(* IEC 61131-3 sources: std_i2980_v2.06_cp053/Source/IMM/ieccontrol/system, 15 files *)

(* ---- ABCfgLoader.pu ---- *)
(*
@h    ! WARNING !
@h    The Kemro K2 system (including software) only meets category B according to EN 954-1,
@h    thus it is not intended for usage in safety-relevant control applications in the field
@h    of personal safety (e.g. emergency stop).
@h    To implement potentially necessary safety-relevant control tasks, always use additional
@h    external safety devices that are intended for the particular purpose, and meet the necessary
@h    functional safety.
@h    For further information see EN 954-1 (EN ISO 13849-1) and/or the K2-x00 user manual, chapter
@h    "CE conformity, directives and standards".

This algorithm block reading configuration settings from
the catalogue and copies the values to the according systemvariables.
Reading starts after device registration is completed.
After reading the settings the file appco.cfg is deleted.
*)

IMPORT_OVER_LISTFILE
 KCAT_GetHandle
, FConfigNode
, KCAT_GetValue
, KFILE_Delete
, FCreateIECVersion
, FCreateIECLibVersion
, FCreateIECBaseVersion
, FCreateSystemName
, FCreateHMIKVSVersion
, FCreateHMIStyleVersion
, KSYS_BPAPI_VAR_TXTREAD
, KCAT_Status_OK
, KCAT_Status
, KSYS_BPApiState
, KCAT_HandleData
, KFILE_Status

END_IMPORT

ALGORITHM_BLOCK ABCfgLoader #DUMMY_EDIT_BLOCK

SYSTEM_VAR
 sv_bReadConfigDone : BOOL;
 sv_bDeviceRegisterDone : BOOL;
 sv_bInitStart : BOOL;
 sv_sPathMasterdisk : STRING(255);
 sv_sPathWorkspace : STRING(255);
 sv_sPathAppldisk : STRING(255);
END_VAR

SYSTEM_OBJECT
 TaskMid : TASK;
 PU_Task_7 : TASK;
 TaskSlow : TASK;
END_OBJECT

FUNCTION fCreateOSVersion : BOOL
 #DUMMY_EDIT_BLOCK

VAR
 Status : KCAT_Status;
 SysState : KSYS_BPApiState;
 HandleData : KCAT_HandleData;
 sValue : STRING(255);
 sTmp : STRING(255);
 bLinux : BOOL;
END_VAR
#BEGIN_EDIT_BLOCK
(**************************************** WARNING ********************************************
 *** The KEBA Kemro K2 System including software is not intended for safety control tasks! ***
 ***                       For further information see Comment tab!                        ***
 *********************************************************************************************)

// create extended OS version information in catalog (on Linux systems only)
// necessary for systems like KVS to access OS specific version info without SysRPC/BPAPI

HandleData := KCAT_GetHandle('UOS.System');
IF HandleData.Status = KCAT_Status_OK THEN
   Status := KCAT_GetValue(Handle := HandleData.Handle, Buffer := sValue);
   IF (sValue = 'Linux') THEN
      bLinux := TRUE;
   END_IF;
END_IF;

IF(NOT bLinux) THEN
   // do not create the nodes on VxWorks - this info does not exist
   RETURN;
END_IF;

HandleData := KCAT_GetHandle('System');
IF HandleData.Status <> KCAT_Status_OK THEN
   RETURN;
END_IF;

HandleData := KCAT_AddDir(HandleData.Handle, 'OS');
IF HandleData.Status <> KCAT_Status_OK THEN
   RETURN;
END_IF;

// add device driver version

SysState := KSYS_BPAPI_VAR_TXTREAD('SYS.HW.OS.driversVersion', sValue);
Status := KCAT_AddValue(HandleData.Handle, "driversVersion", KCAT_Type_STRING, sValue);
IF Status <> KCAT_Status_OK THEN
   RETURN;
END_IF;

// add OS specific version (concated)
SysState := KSYS_BPAPI_VAR_TXTREAD('SYS.HW.OS.osType', sTmp);
sValue := CONCAT(sTmp, ' ');

SysState := KSYS_BPAPI_VAR_TXTREAD('SYS.HW.OS.osVersion', sTmp);
sValue := CONCAT(sValue, sTmp, ' ');

SysState := KSYS_BPAPI_VAR_TXTREAD('SYS.HW.OS.kernelVersion', sTmp);
sValue := CONCAT(sValue, sTmp);

Status := KCAT_AddValue(HandleData.Handle, "osVersion", KCAT_Type_STRING, sValue);
IF Status <> KCAT_Status_OK THEN
   RETURN;
END_IF;

fCreateOSVersion := TRUE;

;#END_EDIT_BLOCK END_FUNCTION

PROCESS_ALGORITHM paReadConfig ON TaskMid

VAR
 HandleData : KCAT_HandleData;
 sRootPath : STRING(255);
 // sPath : STRING(255);
 // Status : KCAT_Status;
 // sBasePath : STRING(255);
 fileState : KFILE_Status;
 StatusName_CAT : KCAT_HandleData;
 Status_CAT : KCAT_Status;
END_VAR
#BEGIN_EDIT_BLOCK
(**************************************** WARNING ********************************************
 *** The KEBA Kemro K2 System including software is not intended for safety control tasks! ***
 ***                       For further information see Comment tab!                        ***
 *********************************************************************************************)

//check if data is available
sRootPath := "Application.Application1";
HandleData:=KCAT_GetHandle(sRootPath);
IF HandleData.Status<>KCAT_Status_OK THEN
   //no catalog entries for appliaction available
   sv_bReadConfigDone := TRUE;
   STOP_PROCESS_ALGORITHM();
   RETURN;
END_IF;

(*
//-----------------------------------------------------------
//read actuation params
//-------------------------------------------------------------
sBasePath := CONCAT(sRootPath, ".Actuation");

sPath := CONCAT(sBasePath, ".System_pressure");
Status := FConfigNode(sPath, "system.sv_rMaximumPressure", 1);

sPath := CONCAT(sBasePath, ".System_velocity");
Status := FConfigNode(sPath, "Injection1.sv_rMaxSpeedFwd", 1);

//-------------------------------------------------------------------
//read clamp side parameters
//-------------------------------------------------------------------
sBasePath := CONCAT(sRootPath, ".Closure_unit");

//mold stroke
sPath := CONCAT(sBasePath, ".Stroke_mold");
Status := FConfigNode(sPath, "Mold1.sv_rMoldStroke", 1);

//profile stages mold close
sPath := CONCAT(sBasePath, ".No_profile_points_mold_close");
Status := FConfigNode(sPath, "Mold1.sv_MoldFwdProfVisSrc.Profile.iNoOfPoints", 0);

//profile stages mold open
sPath := CONCAT(sBasePath, ".No_profile_points_mold_open");
Status := FConfigNode(sPath, "Mold1.sv_MoldBwdProfVis.Profile.iNoOfPoints", 0);

//ejector stroke
sPath := CONCAT(sBasePath, ".Stroke_ejector");
Status := FConfigNode(sPath, "Ejector1.sv_rEjectorStroke", 1);

//profile stages ejector bwd
sPath := CONCAT(sBasePath, ".No_profile_points_ejector_bwd");
Status := FConfigNode(sPath, "Ejector1.sv_EjectorBwdVis.Profile.iNoOfPoints", 0);

//profile stages ejector fwd
sPath := CONCAT(sBasePath, ".No_profile_points_ejector_fwd");
Status := FConfigNode(sPath, "Ejector1.sv_EjectorFwdVis.Profile.iNoOfPoints", 0);

//mold adjust mode
sPath := CONCAT(sBasePath, ".Mold_adjust");
Status := FConfigNode(sPath, "MoldHeight1.sv_MoldHeightAdjustMotor", 3);

//mold heating
sPath := CONCAT(sBasePath, ".No_heating_zones");
Status := FConfigNode(sPath, "HeatingMold1.sv_iNumberOfZones", 2);

//------------------------------------------------------------------------------
//read inject side parameters
//------------------------------------------------------------------------------
sBasePath := CONCAT(sRootPath, ".Injection_Unit.Injection_Unit:0");

//screw stroke
sPath := CONCAT(sBasePath, ".Stroke_screw");
Status := FConfigNode(sPath, "Injection1.sv_rScrewStroke", 1);

//nozzle stroke
sPath := CONCAT(sBasePath, ".Stroke_nozzle");
Status := FConfigNode(sPath, "Nozzle1.sv_rNozzleStroke", 1);

//profile stages inject
sPath := CONCAT(sBasePath, ".No_profile_points_inject");
Status := FConfigNode(sPath, "Injection1.sv_InjectProfVis.Profile.iNoOfPoints", 0);

//profile stages hold
sPath := CONCAT(sBasePath, ".No_profile_points_hold");
Status := FConfigNode(sPath, "Injection1.sv_HoldProfVis.Profile.iNoOfPoints", 0);

//profile stages charge
sPath := CONCAT(sBasePath, ".No_profile_points_charge");
Status := FConfigNode(sPath, "Injection1.sv_PlastProfVis.Profile.iNoOfPoints", 0);

//screw impulses per rotation
sPath := CONCAT(sBasePath, ".No_impulses_rotation");
Status := FConfigNode(sPath, "Injection1.sv_iScrewGain", 2);

//number of heating zones
sPath := CONCAT(sBasePath, ".No_heating_zones");
Status := FConfigNode(sPath, "HeatingNozzle1.sv_iNumberOfZones", 2);

//profile stages nozzle fwd
sPath := CONCAT(sBasePath, ".No_profile_points_nozzle_fwd");
Status := FConfigNode(sPath, "Nozzle1.sv_NozzleFwdProfVis.Profile.iNoOfPoints", 0);

//profile stages nozzle bwd
sPath := CONCAT(sBasePath, ".No_profile_points_nozzle_bwd");
Status := FConfigNode(sPath, "Nozzle1.sv_NozzleBwdProfVis.Profile.iNoOfPoints", 0);

//nozzle movement mode
sPath := CONCAT(sBasePath, ".Movement_Mode");
Status := FConfigNode(sPath, "Nozzle1.sv_MovementMode", 4);
//----------------------------------------------------------------------------------------
*)

//delete configuration file
StatusName_CAT := KCAT_GetHandle('System.applPath');
IF StatusName_CAT.Status = KCAT_Status_OK THEN
    Status_CAT := KCAT_GetValue(Handle := StatusName_CAT.Handle, Buffer := sRootPath);
END_IF;

fileState := KFILE_Delete(Name:= CONCAT(sRootPath,'/application/control/config/appco.cfg'));

sv_bReadConfigDone := TRUE;
STOP_PROCESS_ALGORITHM();

;#END_EDIT_BLOCK END_ALGORITHM

POSTUPDATE_ALGORITHM pDeviceRegisterDone ON PU_Task_7 WITH sv_bDeviceRegisterDone

#BEGIN_EDIT_BLOCK
(**************************************** WARNING ********************************************
 *** The KEBA Kemro K2 System including software is not intended for safety control tasks! ***
 ***                       For further information see Comment tab!                        ***
 *********************************************************************************************)

IF sv_bDeviceRegisterDone THEN
   START_PROCESS_ALGORITHM(paReadConfig);
END_IF;

;#END_EDIT_BLOCK END_ALGORITHM

PROCESS_ALGORITHM paVersionInfo ON TaskSlow AUTOSTART

VAR
 b : BOOL;
END_VAR
#BEGIN_EDIT_BLOCK
(**************************************** WARNING ********************************************
 *** The KEBA Kemro K2 System including software is not intended for safety control tasks! ***
 ***                       For further information see Comment tab!                        ***
 *********************************************************************************************)

b := fCreateOSVersion();
b := FCreateIECVersion();
b := FCreateIECLibVersion();
b := FCreateIECBaseVersion();
b := FCreateHMIKVSVersion();
b := FCreateHMIStyleVersion();
b := FCreateSystemName();

STOP_PROCESS_ALGORITHM();

;#END_EDIT_BLOCK END_ALGORITHM

POSTUPDATE_ALGORITHM pUpdateSysPaths ON PU_Task_7 WITH sv_bInitStart

VAR
 hDataKey : KCAT_HandleData;
 hReadStatus : KCAT_Status;
END_VAR
#BEGIN_EDIT_BLOCK
(**************************************** WARNING ********************************************
 *** The KEBA Kemro K2 System including software is not intended for safety control tasks! ***
 ***                       For further information see Comment tab!                        ***
 *********************************************************************************************)

//Initialize the applPath, workPath and rootPath. The paths have to be read from
//UOS catalog. The paths are used conform to PLC docs (path hierarchy).

hDataKey := KCAT_GetHandle('System.rootPath');
IF hDataKey.Status = KCAT_Status_OK THEN
    hReadStatus := KCAT_GetValue(Handle := hDataKey.Handle, Buffer := sv_sPathMasterdisk);
END_IF;

hDataKey := KCAT_GetHandle('System.applPath');
IF hDataKey.Status = KCAT_Status_OK THEN
    hReadStatus := KCAT_GetValue(Handle := hDataKey.Handle, Buffer := sv_sPathAppldisk);
    IF (hReadStatus <> KCAT_Status_OK) OR LEN(sv_sPathAppldisk) < 1 THEN
       sv_sPathAppldisk := sv_sPathMasterdisk;
    END_IF;
END_IF;

hDataKey := KCAT_GetHandle('System.workPath');
IF hDataKey.Status = KCAT_Status_OK THEN
    hReadStatus := KCAT_GetValue(Handle := hDataKey.Handle, Buffer := sv_sPathWorkspace);
    IF (hReadStatus <> KCAT_Status_OK) OR LEN(sv_sPathWorkspace) < 1 THEN
       sv_sPathWorkspace := sv_sPathAppldisk;
    END_IF;
END_IF;

;#END_EDIT_BLOCK END_ALGORITHM

END_ALGORITHM_BLOCK

#END_OF_IEC_PART

@Puma @IecEditor 6 103 @Pou 25
@@@BEG_Comment@@@
@h    ! WARNING !
@h    The Kemro K2 system (including software) only meets category B according to EN 954-1,
@h    thus it is not intended for usage in safety-relevant control applications in the field
@h    of personal safety (e.g. emergency stop).
@h    To implement potentially necessary safety-relevant control tasks, always use additional
@h    external safety devices that are intended for the particular purpose, and meet the necessary
@h    functional safety.
@h    For further information see EN 954-1 (EN ISO 13849-1) and/or the K2-x00 user manual, chapter
@h    "CE conformity, directives and standards".

This algorithm block reading configuration settings from
the catalogue and copies the values to the according systemvariables.
Reading starts after device registration is completed.
After reading the settings the file appco.cfg is deleted.
@@@END_Comment@@@

@BEG_Contents

@BEG_Func
@RT(17)FuncTreeContainer
11
@Var @RT(14)KCAT_GetHandle @RT(0) @T @T @DERIVED 0 @F @RT(22)KEBA_STANDARD_FUNCTION @F
@T
@BEG_Attrib
0 @RT(0) @RT(0)
@END_Attrib
1 1 @F @F @F @F

@Var @RT(11)FConfigNode @RT(0) @T @T @DERIVED 0 @F @RT(8)FUNCTION @F
@T
@BEG_Attrib
0 @RT(0) @RT(0)
@END_Attrib
1 1 @F @F @F @F

@Var @RT(13)KCAT_GetValue @RT(0) @T @T @DERIVED 0 @F @RT(22)KEBA_STANDARD_FUNCTION @F
@T
@BEG_Attrib
0 @RT(0) @RT(0)
@END_Attrib
1 1 @F @F @F @F

@Var @RT(12)KFILE_Delete @RT(0) @T @T @DERIVED 0 @F @RT(22)KEBA_STANDARD_FUNCTION @F
@T
@BEG_Attrib
0 @RT(0) @RT(0)
@END_Attrib
1 1 @F @F @F @F

@Var @RT(17)FCreateIECVersion @RT(0) @T @T @DERIVED 0 @F @RT(8)FUNCTION @F
@T
@BEG_Attrib
0 @RT(0) @RT(0)
@END_Attrib
1 1 @F @F @F @F

@Var @RT(20)FCreateIECLibVersion @RT(0) @T @T @DERIVED 0 @F @RT(8)FUNCTION @F
@T
@BEG_Attrib
0 @RT(0) @RT(0)
@END_Attrib
1 1 @F @F @F @F

@Var @RT(21)FCreateIECBaseVersion @RT(0) @T @T @DERIVED 0 @F @RT(8)FUNCTION @F
@T
@BEG_Attrib
0 @RT(0) @RT(0)
@END_Attrib
1 1 @F @F @F @F

@Var @RT(17)FCreateSystemName @RT(0) @T @T @DERIVED 0 @F @RT(8)FUNCTION @F
@T
@BEG_Attrib
0 @RT(0) @RT(0)
@END_Attrib
1 1 @F @F @F @F

@Var @RT(20)FCreateHMIKVSVersion @RT(0) @T @T @DERIVED 0 @F @RT(8)FUNCTION @F
@T
@BEG_Attrib
0 @RT(0) @RT(0)
@END_Attrib
1 1 @F @F @F @F

@Var @RT(22)FCreateHMIStyleVersion @RT(0) @T @T @DERIVED 0 @F @RT(8)FUNCTION @F
@T
@BEG_Attrib
0 @RT(0) @RT(0)
@END_Attrib
1 1 @F @F @F @F

@Var @RT(22)KSYS_BPAPI_VAR_TXTREAD @RT(0) @T @T @DERIVED 0 @F @RT(22)KEBA_STANDARD_FUNCTION @F
@T
@BEG_Attrib
0 @RT(0) @RT(0)
@END_Attrib
1 1 @F @F @F @F

@END_Func

@BEG_Const
@RT(18)ConstTreeContainer
1
@Var @RT(14)KCAT_Status_OK @RT(0) @T @T @DERIVED 0 @F @RT(11)KCAT_Status @F
@T
@BEG_Attrib
0 @RT(1)0 @RT(0)
@END_Attrib
1 1 @F @F @F @F

@END_Const

@BEG_Export

@BEG_Kind
@ALGORITHM_BLOCK @RT(11)ABCfgLoader @STRUCTURED_TEXT
@RT(0) @RT(0) @RT(0)
@END_Kind

@BEG_Dcl
@RT(16)DclTreeContainer
9
@Var @RT(18)sv_bReadConfigDone @RT(0) @T @F @DT @RT(4)BOOL @RT(0) @T @T @BASIC 0 @F
@F @F
@T
@BEG_Attrib
3 @RT(0) @RT(0) @RT(0)
@END_Attrib
1 8 @F @F @F @F

@Var @RT(22)sv_bDeviceRegisterDone @RT(0) @T @F @DT @RT(4)BOOL @RT(0) @T @T @BASIC 0 @F
@F @F
@T
@BEG_Attrib
3 @RT(0) @RT(0) @RT(0)
@END_Attrib
1 8 @F @F @F @F

@Var @RT(7)TaskMid @RT(0) @T @F @DT @RT(4)TASK @RT(0) @T @T @BASIC 0 @F
@F @F
@T
@BEG_Attrib
3 @RT(0) @RT(0) @RT(0)
@END_Attrib
1 7 @F @F @F @F

@Var @RT(9)PU_Task_7 @RT(0) @T @F @DT @RT(4)TASK @RT(0) @T @T @BASIC 0 @F
@F @F
@T
@BEG_Attrib
3 @RT(0) @RT(0) @RT(0)
@END_Attrib
1 7 @F @F @F @F

@Var @RT(8)TaskSlow @RT(0) @T @F @DT @RT(4)TASK @RT(0) @T @T @BASIC 0 @F
@F @F
@T
@BEG_Attrib
3 @RT(0) @RT(0) @RT(0)
@END_Attrib
1 7 @F @F @F @F

@Var @RT(13)sv_bInitStart @RT(0) @T @F @DT @RT(4)BOOL @RT(0) @T @T @BASIC 0 @F
@F @F
@T
@BEG_Attrib
3 @RT(0) @RT(0) @RT(0)
@END_Attrib
1 8 @F @F @F @F

@Var @RT(18)sv_sPathMasterdisk @RT(0) @T @F @DT @RT(11)STRING(255) @RT(0) @T @T @STRING 0 @F @RT(3)255 @F
@F @F
@T
@BEG_Attrib
3 @RT(0) @RT(0) @RT(0)
@END_Attrib
1 8 @F @F @F @F

@Var @RT(17)sv_sPathWorkspace @RT(0) @T @F @DT @RT(11)STRING(255) @RT(0) @T @T @STRING 0 @F @RT(3)255 @F
@F @F
@T
@BEG_Attrib
3 @RT(0) @RT(0) @RT(0)
@END_Attrib
1 8 @F @F @F @F

@Var @RT(16)sv_sPathAppldisk @RT(0) @T @F @DT @RT(11)STRING(255) @RT(0) @T @T @STRING 0 @F @RT(3)255 @F
@F @F
@T
@BEG_Attrib
3 @RT(0) @RT(0) @RT(0)
@END_Attrib
1 8 @F @F @F @F

@END_Dcl

@END_Export

@BEG_Body

5

@BEG_Export

@BEG_Algo
@FUNCTION @RT(16)fCreateOSVersion @STRUCTURED_TEXT
@RT(4)BOOL @RT(0) @RT(0) @F @F
@END_Algo

@BEG_Dcl
@RT(16)DclTreeContainer
6
@Var @RT(6)Status @RT(0) @T @T @DERIVED 0 @T @T @DT @RT(11)KCAT_Status @RT(0) @T @T @UNKNOWN 0 @F
@F @F
@T
@BEG_Attrib
3 @RT(0) @RT(0) @RT(0)
@END_Attrib
1 0 @F @F @F @F

@Var @RT(8)SysState @RT(0) @T @T @DERIVED 0 @T @T @DT @RT(15)KSYS_BPApiState @RT(0) @T @T @UNKNOWN 0 @F
@F @F
@T
@BEG_Attrib
3 @RT(0) @RT(0) @RT(0)
@END_Attrib
1 0 @F @F @F @F

@Var @RT(10)HandleData @RT(0) @T @T @DERIVED 0 @T @T @DT @RT(15)KCAT_HandleData @RT(0) @T @T @UNKNOWN 0 @F
@F @F
@T
@BEG_Attrib
3 @RT(0) @RT(0) @RT(0)
@END_Attrib
1 0 @F @F @F @F

@Var @RT(6)sValue @RT(0) @T @F @DT @RT(11)STRING(255) @RT(0) @T @T @STRING 0 @F @RT(3)255 @F
@F @F
@T
@BEG_Attrib
3 @RT(0) @RT(0) @RT(0)
@END_Attrib
1 0 @F @F @F @F

@Var @RT(4)sTmp @RT(0) @T @F @DT @RT(11)STRING(255) @RT(0) @T @T @STRING 0 @F @RT(3)255 @F
@F @F
@T
@BEG_Attrib
3 @RT(0) @RT(0) @RT(0)
@END_Attrib
1 0 @F @F @F @F

@Var @RT(6)bLinux @RT(0) @T @F @DT @RT(4)BOOL @RT(0) @T @T @BASIC 0 @F
@F @F
@T
@BEG_Attrib
3 @RT(0) @RT(0) @RT(0)
@END_Attrib
1 0 @F @F @F @F

@END_Dcl

@END_Export

@BEG_Export

@BEG_Algo
@PROCESS_ALGORITHM @RT(12)paReadConfig @STRUCTURED_TEXT
@RT(0) @RT(0) @RT(7)TaskMid @F @F
@END_Algo

@BEG_Dcl
@RT(16)DclTreeContainer
8
@Var @RT(10)HandleData @RT(0) @T @T @DERIVED 0 @T @T @DT @RT(15)KCAT_HandleData @RT(0) @T @T @UNKNOWN 0 @F
@F @F
@T
@BEG_Attrib
3 @RT(0) @RT(0) @RT(0)
@END_Attrib
1 0 @F @F @F @F

@Var @RT(9)sRootPath @RT(0) @T @F @DT @RT(11)STRING(255) @RT(0) @T @T @STRING 0 @F @RT(3)255 @F
@F @F
@T
@BEG_Attrib
3 @RT(0) @RT(0) @RT(0)
@END_Attrib
1 0 @F @F @F @F

@Var @RT(5)sPath @RT(0) @T @F @DT @RT(11)STRING(255) @RT(0) @T @T @STRING 0 @F @RT(3)255 @F
@F @T
@T
@BEG_Attrib
3 @RT(0) @RT(0) @RT(0)
@END_Attrib
1 0 @F @F @F @F

@Var @RT(6)Status @RT(0) @T @T @DERIVED 0 @T @T @DT @RT(11)KCAT_Status @RT(0) @T @T @UNKNOWN 0 @F
@F @T
@T
@BEG_Attrib
3 @RT(0) @RT(0) @RT(0)
@END_Attrib
1 0 @F @F @F @F

@Var @RT(9)sBasePath @RT(0) @T @F @DT @RT(11)STRING(255) @RT(0) @T @T @STRING 0 @F @RT(3)255 @F
@F @T
@T
@BEG_Attrib
3 @RT(0) @RT(0) @RT(0)
@END_Attrib
1 0 @F @F @F @F

@Var @RT(9)fileState @RT(0) @T @T @DERIVED 0 @T @T @DT @RT(12)KFILE_Status @RT(0) @T @T @UNKNOWN 0 @F
@F @F
@T
@BEG_Attrib
3 @RT(0) @RT(0) @RT(0)
@END_Attrib
1 0 @F @F @F @F

@Var @RT(14)StatusName_CAT @RT(0) @T @T @DERIVED 0 @T @T @DT @RT(15)KCAT_HandleData @RT(0) @T @T @UNKNOWN 0 @F
@F @F
@T
@BEG_Attrib
3 @RT(0) @RT(0) @RT(0)
@END_Attrib
1 0 @F @F @F @F

@Var @RT(10)Status_CAT @RT(0) @T @T @DERIVED 0 @T @T @DT @RT(11)KCAT_Status @RT(0) @T @T @UNKNOWN 0 @F
@F @F
@T
@BEG_Attrib
3 @RT(0) @RT(0) @RT(0)
@END_Attrib
1 0 @F @F @F @F

@END_Dcl

@END_Export

@BEG_Export

@BEG_Algo
@POSTUPDATE_ALGORITHM @RT(19)pDeviceRegisterDone @STRUCTURED_TEXT
@RT(0) @RT(22)sv_bDeviceRegisterDone @RT(9)PU_Task_7 @F @F
@END_Algo

@BEG_Dcl
@RT(16)DclTreeContainer
0
@END_Dcl

@END_Export

@BEG_Export

@BEG_Algo
@PROCESS_ALGORITHM @RT(13)paVersionInfo @STRUCTURED_TEXT
@RT(0) @RT(0) @RT(8)TaskSlow @T @F
@END_Algo

@BEG_Dcl
@RT(16)DclTreeContainer
1
@Var @RT(1)b @RT(0) @T @F @DT @RT(4)BOOL @RT(0) @T @T @BASIC 0 @F
@F @F
@T
@BEG_Attrib
3 @RT(0) @RT(0) @RT(0)
@END_Attrib
1 0 @F @F @F @F

@END_Dcl

@END_Export

@BEG_Export

@BEG_Algo
@POSTUPDATE_ALGORITHM @RT(15)pUpdateSysPaths @STRUCTURED_TEXT
@RT(0) @RT(13)sv_bInitStart @RT(9)PU_Task_7 @F @F
@END_Algo

@BEG_Dcl
@RT(16)DclTreeContainer
2
@Var @RT(8)hDataKey @RT(0) @T @T @DERIVED 0 @T @T @DT @RT(15)KCAT_HandleData @RT(0) @T @T @UNKNOWN 0 @F
@F @F
@T
@BEG_Attrib
3 @RT(0) @RT(0) @RT(0)
@END_Attrib
1 0 @F @F @F @F

@Var @RT(11)hReadStatus @RT(0) @T @T @DERIVED 0 @T @T @DT @RT(11)KCAT_Status @RT(0) @T @T @UNKNOWN 0 @F
@F @F
@T
@BEG_Attrib
3 @RT(0) @RT(0) @RT(0)
@END_Attrib
1 0 @F @F @F @F

@END_Dcl

@END_Export

@BEG_Body
@TL(57)
(**************************************** WARNING ********************************************
 *** The KEBA Kemro K2 System including software is not intended for safety control tasks! ***
 ***                       For further information see Comment tab!                        ***
 *********************************************************************************************)

// create extended OS version information in catalog (on Linux systems only)
// necessary for systems like KVS to access OS specific version info without SysRPC/BPAPI

HandleData := KCAT_GetHandle('UOS.System');
IF HandleData.Status = KCAT_Status_OK THEN
   Status := KCAT_GetValue(Handle := HandleData.Handle, Buffer := sValue);
   IF (sValue = 'Linux') THEN
      bLinux := TRUE;
   END_IF;
END_IF;

IF(NOT bLinux) THEN
   // do not create the nodes on VxWorks - this info does not exist
   RETURN;
END_IF;

HandleData := KCAT_GetHandle('System');
IF HandleData.Status <> KCAT_Status_OK THEN
   RETURN;
END_IF;

HandleData := KCAT_AddDir(HandleData.Handle, 'OS');
IF HandleData.Status <> KCAT_Status_OK THEN
   RETURN;
END_IF;

// add device driver version

SysState := KSYS_BPAPI_VAR_TXTREAD('SYS.HW.OS.driversVersion', sValue);
Status := KCAT_AddValue(HandleData.Handle, "driversVersion", KCAT_Type_STRING, sValue);
IF Status <> KCAT_Status_OK THEN
   RETURN;
END_IF;

// add OS specific version (concated)
SysState := KSYS_BPAPI_VAR_TXTREAD('SYS.HW.OS.osType', sTmp);
sValue := CONCAT(sTmp, ' ');

SysState := KSYS_BPAPI_VAR_TXTREAD('SYS.HW.OS.osVersion', sTmp);
sValue := CONCAT(sValue, sTmp, ' ');

SysState := KSYS_BPAPI_VAR_TXTREAD('SYS.HW.OS.kernelVersion', sTmp);
sValue := CONCAT(sValue, sTmp);

Status := KCAT_AddValue(HandleData.Handle, "osVersion", KCAT_Type_STRING, sValue);
IF Status <> KCAT_Status_OK THEN
   RETURN;
END_IF;

fCreateOSVersion := TRUE;

@END_Body

@@@BEG_Comment@@@
@TL(0)

@@@END_Comment@@@

@BEG_Body
@TL(124)
(**************************************** WARNING ********************************************
 *** The KEBA Kemro K2 System including software is not intended for safety control tasks! ***
 ***                       For further information see Comment tab!                        ***
 *********************************************************************************************)

//check if data is available
sRootPath := "Application.Application1";
HandleData:=KCAT_GetHandle(sRootPath);
IF HandleData.Status<>KCAT_Status_OK THEN
   //no catalog entries for appliaction available
   sv_bReadConfigDone := TRUE;
   STOP_PROCESS_ALGORITHM();
   RETURN;
END_IF;

(*
//-----------------------------------------------------------
//read actuation params
//-------------------------------------------------------------
sBasePath := CONCAT(sRootPath, ".Actuation");

sPath := CONCAT(sBasePath, ".System_pressure");
Status := FConfigNode(sPath, "system.sv_rMaximumPressure", 1);

sPath := CONCAT(sBasePath, ".System_velocity");
Status := FConfigNode(sPath, "Injection1.sv_rMaxSpeedFwd", 1);

//-------------------------------------------------------------------
//read clamp side parameters
//-------------------------------------------------------------------
sBasePath := CONCAT(sRootPath, ".Closure_unit");

//mold stroke
sPath := CONCAT(sBasePath, ".Stroke_mold");
Status := FConfigNode(sPath, "Mold1.sv_rMoldStroke", 1);

//profile stages mold close
sPath := CONCAT(sBasePath, ".No_profile_points_mold_close");
Status := FConfigNode(sPath, "Mold1.sv_MoldFwdProfVisSrc.Profile.iNoOfPoints", 0);

//profile stages mold open
sPath := CONCAT(sBasePath, ".No_profile_points_mold_open");
Status := FConfigNode(sPath, "Mold1.sv_MoldBwdProfVis.Profile.iNoOfPoints", 0);

//ejector stroke
sPath := CONCAT(sBasePath, ".Stroke_ejector");
Status := FConfigNode(sPath, "Ejector1.sv_rEjectorStroke", 1);

//profile stages ejector bwd
sPath := CONCAT(sBasePath, ".No_profile_points_ejector_bwd");
Status := FConfigNode(sPath, "Ejector1.sv_EjectorBwdVis.Profile.iNoOfPoints", 0);

//profile stages ejector fwd
sPath := CONCAT(sBasePath, ".No_profile_points_ejector_fwd");
Status := FConfigNode(sPath, "Ejector1.sv_EjectorFwdVis.Profile.iNoOfPoints", 0);

//mold adjust mode
sPath := CONCAT(sBasePath, ".Mold_adjust");
Status := FConfigNode(sPath, "MoldHeight1.sv_MoldHeightAdjustMotor", 3);

//mold heating
sPath := CONCAT(sBasePath, ".No_heating_zones");
Status := FConfigNode(sPath, "HeatingMold1.sv_iNumberOfZones", 2);

//------------------------------------------------------------------------------
//read inject side parameters
//------------------------------------------------------------------------------
sBasePath := CONCAT(sRootPath, ".Injection_Unit.Injection_Unit:0");

//screw stroke
sPath := CONCAT(sBasePath, ".Stroke_screw");
Status := FConfigNode(sPath, "Injection1.sv_rScrewStroke", 1);

//nozzle stroke
sPath := CONCAT(sBasePath, ".Stroke_nozzle");
Status := FConfigNode(sPath, "Nozzle1.sv_rNozzleStroke", 1);

//profile stages inject
sPath := CONCAT(sBasePath, ".No_profile_points_inject");
Status := FConfigNode(sPath, "Injection1.sv_InjectProfVis.Profile.iNoOfPoints", 0);

//profile stages hold
sPath := CONCAT(sBasePath, ".No_profile_points_hold");
Status := FConfigNode(sPath, "Injection1.sv_HoldProfVis.Profile.iNoOfPoints", 0);

//profile stages charge
sPath := CONCAT(sBasePath, ".No_profile_points_charge");
Status := FConfigNode(sPath, "Injection1.sv_PlastProfVis.Profile.iNoOfPoints", 0);

//screw impulses per rotation
sPath := CONCAT(sBasePath, ".No_impulses_rotation");
Status := FConfigNode(sPath, "Injection1.sv_iScrewGain", 2);

//number of heating zones
sPath := CONCAT(sBasePath, ".No_heating_zones");
Status := FConfigNode(sPath, "HeatingNozzle1.sv_iNumberOfZones", 2);

//profile stages nozzle fwd
sPath := CONCAT(sBasePath, ".No_profile_points_nozzle_fwd");
Status := FConfigNode(sPath, "Nozzle1.sv_NozzleFwdProfVis.Profile.iNoOfPoints", 0);

//profile stages nozzle bwd
sPath := CONCAT(sBasePath, ".No_profile_points_nozzle_bwd");
Status := FConfigNode(sPath, "Nozzle1.sv_NozzleBwdProfVis.Profile.iNoOfPoints", 0);

//nozzle movement mode
sPath := CONCAT(sBasePath, ".Movement_Mode");
Status := FConfigNode(sPath, "Nozzle1.sv_MovementMode", 4);
//----------------------------------------------------------------------------------------
*)

//delete configuration file
StatusName_CAT := KCAT_GetHandle('System.applPath');
IF StatusName_CAT.Status = KCAT_Status_OK THEN
    Status_CAT := KCAT_GetValue(Handle := StatusName_CAT.Handle, Buffer := sRootPath);
END_IF;

fileState := KFILE_Delete(Name:= CONCAT(sRootPath,'/application/control/config/appco.cfg'));

sv_bReadConfigDone := TRUE;
STOP_PROCESS_ALGORITHM();

@END_Body

@@@BEG_Comment@@@
@TL(0)

@@@END_Comment@@@

@BEG_Body
@TL(9)
(**************************************** WARNING ********************************************
 *** The KEBA Kemro K2 System including software is not intended for safety control tasks! ***
 ***                       For further information see Comment tab!                        ***
 *********************************************************************************************)

IF sv_bDeviceRegisterDone THEN
   START_PROCESS_ALGORITHM(paReadConfig);
END_IF;

@END_Body

@@@BEG_Comment@@@
@TL(0)

@@@END_Comment@@@

@BEG_Body
@TL(16)
(**************************************** WARNING ********************************************
 *** The KEBA Kemro K2 System including software is not intended for safety control tasks! ***
 ***                       For further information see Comment tab!                        ***
 *********************************************************************************************)

b := fCreateOSVersion();
b := FCreateIECVersion();
b := FCreateIECLibVersion();
b := FCreateIECBaseVersion();
b := FCreateHMIKVSVersion();
b := FCreateHMIStyleVersion();
b := FCreateSystemName();

STOP_PROCESS_ALGORITHM();

@END_Body

@@@BEG_Comment@@@
@TL(0)

@@@END_Comment@@@

@BEG_Body
@TL(32)
(**************************************** WARNING ********************************************
 *** The KEBA Kemro K2 System including software is not intended for safety control tasks! ***
 ***                       For further information see Comment tab!                        ***
 *********************************************************************************************)

//Initialize the applPath, workPath and rootPath. The paths have to be read from
//UOS catalog. The paths are used conform to PLC docs (path hierarchy).

hDataKey := KCAT_GetHandle('System.rootPath');
IF hDataKey.Status = KCAT_Status_OK THEN
    hReadStatus := KCAT_GetValue(Handle := hDataKey.Handle, Buffer := sv_sPathMasterdisk);
END_IF;

hDataKey := KCAT_GetHandle('System.applPath');
IF hDataKey.Status = KCAT_Status_OK THEN
    hReadStatus := KCAT_GetValue(Handle := hDataKey.Handle, Buffer := sv_sPathAppldisk);
    IF (hReadStatus <> KCAT_Status_OK) OR LEN(sv_sPathAppldisk) < 1 THEN
       sv_sPathAppldisk := sv_sPathMasterdisk;
    END_IF;
END_IF;

hDataKey := KCAT_GetHandle('System.workPath');
IF hDataKey.Status = KCAT_Status_OK THEN
    hReadStatus := KCAT_GetValue(Handle := hDataKey.Handle, Buffer := sv_sPathWorkspace);
    IF (hReadStatus <> KCAT_Status_OK) OR LEN(sv_sPathWorkspace) < 1 THEN
       sv_sPathWorkspace := sv_sPathAppldisk;
    END_IF;
END_IF;

@END_Body

@@@BEG_Comment@@@
@TL(0)

@@@END_Comment@@@
@END_Body

@END_Contents

(* ---- FConfigNode.pu ---- *)
(*
@h    ! WARNING !
@h    The Kemro K2 system (including software) only meets category B according to EN 954-1,
@h    thus it is not intended for usage in safety-relevant control applications in the field
@h    of personal safety (e.g. emergency stop).
@h    To implement potentially necessary safety-relevant control tasks, always use additional
@h    external safety devices that are intended for the particular purpose, and meet the necessary
@h    functional safety.
@h    For further information see EN 954-1 (EN ISO 13849-1) and/or the K2-x00 user manual, chapter
@h    "CE conformity, directives and standards".

*)

IMPORT_OVER_LISTFILE
 KCAT_GetValue
, KCAT_Status
, KSYS_Status
, KCAT_HandleData
, tnMotorType
, tnMovementMode

END_IMPORT

FUNCTION FConfigNode : KCAT_Status #DUMMY_EDIT_BLOCK

VAR_INPUT
 sPath : STRING(255);
 sSVName : STRING(255);
 iType : DINT (* datatype (0:UDINT, 1:REAL, 2:DINT) *);
END_VAR

VAR
 st : KSYS_Status;
 puValue : REFTO UDINT;
 prValue : REFTO REAL;
 piValue : REFTO DINT;
 HandleData : KCAT_HandleData;
 Status : KCAT_Status;
 uValue : UDINT;
 rValue : LREAL;
 iValue : DINT;
 pMoldAdjMotorType : REFTO tnMotorType;
 pNozzleMovementMode : REFTO tnMovementMode;
END_VAR
#BEGIN_EDIT_BLOCK

HandleData:=KCAT_GetHandle(sPath);
IF HandleData.Status<>KCAT_Status_OK THEN
  RETURN;
END_IF;

CASE iType OF

   0: // UDINT
     Status:=KCAT_GetValue(HandleData.Handle, uValue);
     IF Status = KCAT_Status_OK THEN
         puValue := GET_SYNC_REFTO(sSVName, T#0s, st);
         IF st = KSYS_Status_OK THEN
            puValue^:=uValue;
         END_IF;
     END_IF;

   1: // REAL
     Status:=KCAT_GetValue(HandleData.Handle, rValue);
     IF Status = KCAT_Status_OK THEN
         prValue:=GET_SYNC_REFTO(sSVName, T#0s, st);
         IF st = KSYS_Status_OK THEN
            prValue^:=LREAL_TO_REAL(rValue);
         END_IF;
     END_IF;

   2: // DINT
     Status:=KCAT_GetValue(HandleData.Handle, iValue);
     IF Status = KCAT_Status_OK THEN
         piValue := GET_SYNC_REFTO(sSVName, T#0s, st);
         IF st = KSYS_Status_OK THEN
            piValue^:=iValue;
         END_IF;
     END_IF;

   3: // tnMotorType (mold adjust motor type)
     Status:=KCAT_GetValue(HandleData.Handle, iValue);
     IF Status = KCAT_Status_OK THEN
         pMoldAdjMotorType := GET_SYNC_REFTO(sSVName, T#0s, st);
         IF st = KSYS_Status_OK THEN
            IF iValue = 0 THEN
               pMoldAdjMotorType^ := nHydraulic; //hydraulic mold adjust motor
            ELSIF iValue = 1 THEN
               pMoldAdjMotorType^ := nElectric; //electric mold adjust motor;
            END_IF;
         END_IF;
      END_IF;

   4: // tnMovementMode (nozzle movement mode)
     Status:=KCAT_GetValue(HandleData.Handle, iValue);
     IF Status = KCAT_Status_OK THEN
           pNozzleMovementMode := GET_SYNC_REFTO(sSVName, T#0s, st);
           IF st = KSYS_Status_OK THEN
              IF iValue = 0 THEN
                 pNozzleMovementMode^ := nPositionDependent; //position dependent
              ELSIF iValue = 1 THEN
                 pNozzleMovementMode^ := nLimitSwitchDependent; //limit switch dependent;
              ELSIF iValue = 2 THEN
                 pNozzleMovementMode^ := nMoveTimeDependent; //time dependent;
              END_IF;
           END_IF;
      END_IF;

ELSE
   ;
END_CASE;

FConfigNode:=Status;

;#END_EDIT_BLOCK END_FUNCTION

#END_OF_IEC_PART

@Puma @IecEditor 6 68 @Pou 25
@@@BEG_Comment@@@
@h    ! WARNING !
@h    The Kemro K2 system (including software) only meets category B according to EN 954-1,
@h    thus it is not intended for usage in safety-relevant control applications in the field
@h    of personal safety (e.g. emergency stop).
@h    To implement potentially necessary safety-relevant control tasks, always use additional
@h    external safety devices that are intended for the particular purpose, and meet the necessary
@h    functional safety.
@h    For further information see EN 954-1 (EN ISO 13849-1) and/or the K2-x00 user manual, chapter
@h    "CE conformity, directives and standards".

@@@END_Comment@@@

@BEG_Contents

@BEG_Func
@RT(17)FuncTreeContainer
1
@Var @RT(13)KCAT_GetValue @RT(0) @T @T @DERIVED 0 @F @RT(22)KEBA_STANDARD_FUNCTION @F
@T
@BEG_Attrib
0 @RT(0) @RT(0)
@END_Attrib
1 1 @F @F @F @F

@END_Func

@BEG_Const
@RT(18)ConstTreeContainer
0
@END_Const

@BEG_Export

@BEG_Kind
@FUNCTION @RT(11)FConfigNode @STRUCTURED_TEXT
@RT(11)KCAT_Status @RT(0) @RT(0)
@END_Kind

@BEG_Dcl
@RT(16)DclTreeContainer
14
@Var @RT(5)sPath @RT(0) @T @F @DT @RT(11)STRING(255) @RT(0) @T @T @STRING 0 @F @RT(3)255 @F
@F @F
@T
@BEG_Attrib
3 @RT(0) @RT(0) @RT(0)
@END_Attrib
1 1 @F @F @F @F

@Var @RT(7)sSVName @RT(0) @T @F @DT @RT(11)STRING(255) @RT(0) @T @T @STRING 0 @F @RT(3)255 @F
@F @F
@T
@BEG_Attrib
3 @RT(0) @RT(0) @RT(0)
@END_Attrib
1 1 @F @F @F @F

@Var @RT(5)iType @RT(0) @T @F @DT @RT(4)DINT @RT(0) @T @T @BASIC 0 @F
@F @F
@T
@BEG_Attrib
3 @RT(0) @RT(34)datatype (0:UDINT, 1:REAL, 2:DINT) @RT(0)
@END_Attrib
1 1 @F @F @F @F

@Var @RT(2)st @RT(0) @T @T @DERIVED 0 @T @T @DT @RT(11)KSYS_Status @RT(0) @T @T @UNKNOWN 0 @F
@F @F
@T
@BEG_Attrib
3 @RT(0) @RT(0) @RT(0)
@END_Attrib
1 0 @F @F @F @F

@Var @RT(7)puValue @RT(0) @T @T @REFTO 0 @T @DT @RT(5)UDINT @RT(0) @T @T @BASIC 0 @F
@F @F
@T
@BEG_Attrib
3 @RT(0) @RT(0) @RT(0)
@END_Attrib
1 0 @F @F @F @F

@Var @RT(7)prValue @RT(0) @T @T @REFTO 0 @T @DT @RT(4)REAL @RT(0) @T @T @BASIC 0 @F
@F @F
@T
@BEG_Attrib
3 @RT(0) @RT(0) @RT(0)
@END_Attrib
1 0 @F @F @F @F

@Var @RT(7)piValue @RT(0) @T @T @REFTO 0 @T @DT @RT(4)DINT @RT(0) @T @T @BASIC 0 @F
@F @F
@T
@BEG_Attrib
3 @RT(0) @RT(0) @RT(0)
@END_Attrib
1 0 @F @F @F @F

@Var @RT(10)HandleData @RT(0) @T @T @DERIVED 0 @T @T @DT @RT(15)KCAT_HandleData @RT(0) @T @T @UNKNOWN 0 @F
@F @F
@T
@BEG_Attrib
3 @RT(0) @RT(0) @RT(0)
@END_Attrib
1 0 @F @F @F @F

@Var @RT(6)Status @RT(0) @T @T @DERIVED 0 @T @T @DT @RT(11)KCAT_Status @RT(0) @T @T @UNKNOWN 0 @F
@F @F
@T
@BEG_Attrib
3 @RT(0) @RT(0) @RT(0)
@END_Attrib
1 0 @F @F @F @F

@Var @RT(6)uValue @RT(0) @T @F @DT @RT(5)UDINT @RT(0) @T @T @BASIC 0 @F
@F @F
@T
@BEG_Attrib
3 @RT(0) @RT(0) @RT(0)
@END_Attrib
1 0 @F @F @F @F

@Var @RT(6)rValue @RT(0) @T @F @DT @RT(5)LREAL @RT(0) @T @T @BASIC 0 @F
@F @F
@T
@BEG_Attrib
3 @RT(0) @RT(0) @RT(0)
@END_Attrib
1 0 @F @F @F @F

@Var @RT(6)iValue @RT(0) @T @F @DT @RT(4)DINT @RT(0) @T @T @BASIC 0 @F
@F @F
@T
@BEG_Attrib
3 @RT(0) @RT(0) @RT(0)
@END_Attrib
1 0 @F @F @F @F

@Var @RT(17)pMoldAdjMotorType @RT(0) @T @T @REFTO 0 @F @DERIVED 0 @T @T @DT @RT(11)tnMotorType @RT(0) @T @T @UNKNOWN 0 @F
@F @F
@T
@BEG_Attrib
3 @RT(0) @RT(0) @RT(0)
@END_Attrib
1 0 @F @F @F @F

@Var @RT(19)pNozzleMovementMode @RT(0) @T @T @REFTO 0 @F @DERIVED 0 @T @T @DT @RT(14)tnMovementMode @RT(0) @T @T @UNKNOWN 0 @F
@F @F
@T
@BEG_Attrib
3 @RT(0) @RT(0) @RT(0)
@END_Attrib
1 0 @F @F @F @F

@END_Dcl

@END_Export

@BEG_Body
@TL(69)

HandleData:=KCAT_GetHandle(sPath);
IF HandleData.Status<>KCAT_Status_OK THEN
  RETURN;
END_IF;

CASE iType OF

   0: // UDINT
     Status:=KCAT_GetValue(HandleData.Handle, uValue);
     IF Status = KCAT_Status_OK THEN
         puValue := GET_SYNC_REFTO(sSVName, T#0s, st);
         IF st = KSYS_Status_OK THEN
            puValue^:=uValue;
         END_IF;
     END_IF;

   1: // REAL
     Status:=KCAT_GetValue(HandleData.Handle, rValue);
     IF Status = KCAT_Status_OK THEN
         prValue:=GET_SYNC_REFTO(sSVName, T#0s, st);
         IF st = KSYS_Status_OK THEN
            prValue^:=LREAL_TO_REAL(rValue);
         END_IF;
     END_IF;

   2: // DINT
     Status:=KCAT_GetValue(HandleData.Handle, iValue);
     IF Status = KCAT_Status_OK THEN
         piValue := GET_SYNC_REFTO(sSVName, T#0s, st);
         IF st = KSYS_Status_OK THEN
            piValue^:=iValue;
         END_IF;
     END_IF;

   3: // tnMotorType (mold adjust motor type)
     Status:=KCAT_GetValue(HandleData.Handle, iValue);
     IF Status = KCAT_Status_OK THEN
         pMoldAdjMotorType := GET_SYNC_REFTO(sSVName, T#0s, st);
         IF st = KSYS_Status_OK THEN
            IF iValue = 0 THEN
               pMoldAdjMotorType^ := nHydraulic; //hydraulic mold adjust motor
            ELSIF iValue = 1 THEN
               pMoldAdjMotorType^ := nElectric; //electric mold adjust motor;
            END_IF;
         END_IF;
      END_IF;

   4: // tnMovementMode (nozzle movement mode)
     Status:=KCAT_GetValue(HandleData.Handle, iValue);
     IF Status = KCAT_Status_OK THEN
           pNozzleMovementMode := GET_SYNC_REFTO(sSVName, T#0s, st);
           IF st = KSYS_Status_OK THEN
              IF iValue = 0 THEN
                 pNozzleMovementMode^ := nPositionDependent; //position dependent
              ELSIF iValue = 1 THEN
                 pNozzleMovementMode^ := nLimitSwitchDependent; //limit switch dependent;
              ELSIF iValue = 2 THEN
                 pNozzleMovementMode^ := nMoveTimeDependent; //time dependent;
              END_IF;
           END_IF;
      END_IF;

ELSE
   ;
END_CASE;

FConfigNode:=Status;

@END_Body

@END_Contents
@@@BEG_Password@@@
M2hzZmhrMw==
@@@END_Password@@@

(* ---- FCreateHMIKVSVersion.pu ---- *)
(*
@h    ! WARNING !
@h    The Kemro K2 system (including software) only meets category B according to EN 954-1,
@h    thus it is not intended for usage in safety-relevant control applications in the field
@h    of personal safety (e.g. emergency stop).
@h    To implement potentially necessary safety-relevant control tasks, always use additional
@h    external safety devices that are intended for the particular purpose, and meet the necessary
@h    functional safety.
@h    For further information see EN 954-1 (EN ISO 13849-1) and/or the K2-x00 user manual, chapter
@h    "CE conformity, directives and standards".

Create empty catalog entry for KVS version info because there is no possibility to create catalog nodes
in KVS. Version Info will be written by KVS at startup.
*)

IMPORT_OVER_LISTFILE
 FWriteComponentVersion

END_IMPORT

FUNCTION FCreateHMIKVSVersion : BOOL #DUMMY_EDIT_BLOCK

VAR CONSTANT
 sComponentName : STRING(255) := 'KePlast.HMI.KVS';
 iComponentNumber : DINT := 0;
 sVersionString : STRING(255) := '';
 iVersionMajor : DINT := 0;
 iVersionMinor : DINT := 0;
END_VAR
#BEGIN_EDIT_BLOCK
(**************************************** WARNING ********************************************
 *** The KEBA Kemro K2 System including software is not intended for safety control tasks! ***
 ***                       For further information see Comment tab!                        ***
 *********************************************************************************************)

FCreateHMIKVSVersion := FWriteComponentVersion(
        sComponentName,
        iComponentNumber,
        sVersionString,
        iVersionMajor,
        iVersionMinor
);

;#END_EDIT_BLOCK END_FUNCTION

#END_OF_IEC_PART

@Puma @IecEditor 6 68 @Pou 25
@@@BEG_Comment@@@
@h    ! WARNING !
@h    The Kemro K2 system (including software) only meets category B according to EN 954-1,
@h    thus it is not intended for usage in safety-relevant control applications in the field
@h    of personal safety (e.g. emergency stop).
@h    To implement potentially necessary safety-relevant control tasks, always use additional
@h    external safety devices that are intended for the particular purpose, and meet the necessary
@h    functional safety.
@h    For further information see EN 954-1 (EN ISO 13849-1) and/or the K2-x00 user manual, chapter
@h    "CE conformity, directives and standards".

Create empty catalog entry for KVS version info because there is no possibility to create catalog nodes
in KVS. Version Info will be written by KVS at startup.
@@@END_Comment@@@

@BEG_Contents

@BEG_Func
@RT(17)FuncTreeContainer
1
@Var @RT(22)FWriteComponentVersion @RT(0) @T @T @DERIVED 0 @F @RT(8)FUNCTION @F
@T
@BEG_Attrib
0 @RT(0) @RT(0)
@END_Attrib
1 1 @F @F @F @F

@END_Func

@BEG_Const
@RT(18)ConstTreeContainer
0
@END_Const

@BEG_Export

@BEG_Kind
@FUNCTION @RT(20)FCreateHMIKVSVersion @STRUCTURED_TEXT
@RT(4)BOOL @RT(0) @RT(0)
@END_Kind

@BEG_Dcl
@RT(16)DclTreeContainer
5
@Var @RT(14)sComponentName @RT(0) @T @F @DT @RT(11)STRING(255) @RT(0) @T @T @STRING 0 @F @RT(3)255 @F
@F @F
@T
@BEG_Attrib
3 @RT(17)'KePlast.HMI.KVS' @RT(0) @RT(0)
@END_Attrib
1 15 @F @F @F @F

@Var @RT(16)iComponentNumber @RT(0) @T @F @DT @RT(4)DINT @RT(0) @T @T @BASIC 0 @F
@F @F
@T
@BEG_Attrib
3 @RT(1)0 @RT(0) @RT(0)
@END_Attrib
1 15 @F @F @F @F

@Var @RT(14)sVersionString @RT(0) @T @F @DT @RT(11)STRING(255) @RT(0) @T @T @STRING 0 @F @RT(3)255 @F
@F @F
@T
@BEG_Attrib
3 @RT(2)'' @RT(0) @RT(0)
@END_Attrib
1 15 @F @F @F @F

@Var @RT(13)iVersionMajor @RT(0) @T @F @DT @RT(4)DINT @RT(0) @T @T @BASIC 0 @F
@F @F
@T
@BEG_Attrib
3 @RT(1)0 @RT(0) @RT(0)
@END_Attrib
1 15 @F @F @F @F

@Var @RT(13)iVersionMinor @RT(0) @T @F @DT @RT(4)DINT @RT(0) @T @T @BASIC 0 @F
@F @F
@T
@BEG_Attrib
3 @RT(1)0 @RT(0) @RT(0)
@END_Attrib
1 15 @F @F @F @F

@END_Dcl

@END_Export

@BEG_Body
@TL(13)
(**************************************** WARNING ********************************************
 *** The KEBA Kemro K2 System including software is not intended for safety control tasks! ***
 ***                       For further information see Comment tab!                        ***
 *********************************************************************************************)

FCreateHMIKVSVersion := FWriteComponentVersion(
        sComponentName,
        iComponentNumber,
        sVersionString,
        iVersionMajor,
        iVersionMinor
);

@END_Body

@END_Contents

(* ---- FCreateHMIStyleVersion.pu ---- *)
(*
@h    ! WARNING !
@h    The Kemro K2 system (including software) only meets category B according to EN 954-1,
@h    thus it is not intended for usage in safety-relevant control applications in the field
@h    of personal safety (e.g. emergency stop).
@h    To implement potentially necessary safety-relevant control tasks, always use additional
@h    external safety devices that are intended for the particular purpose, and meet the necessary
@h    functional safety.
@h    For further information see EN 954-1 (EN ISO 13849-1) and/or the K2-x00 user manual, chapter
@h    "CE conformity, directives and standards".

Create empty catalog entry for HMI.Style version info because there is no possibility to create catalog nodes
in HMI.Style. Version Info will be written by HMI.Style at startup.
*)

IMPORT_OVER_LISTFILE
 FWriteComponentVersion

END_IMPORT

FUNCTION FCreateHMIStyleVersion : BOOL #DUMMY_EDIT_BLOCK

VAR CONSTANT
 sComponentName : STRING(255) := 'KePlast.HMI.Style';
 iComponentNumber : DINT := 0;
 sVersionString : STRING(255) := '';
 iVersionMajor : DINT := 0;
 iVersionMinor : DINT := 0;
END_VAR
#BEGIN_EDIT_BLOCK
(**************************************** WARNING ********************************************
 *** The KEBA Kemro K2 System including software is not intended for safety control tasks! ***
 ***                       For further information see Comment tab!                        ***
 *********************************************************************************************)

FCreateHMIStyleVersion := FWriteComponentVersion(
        sComponentName,
        iComponentNumber,
        sVersionString,
        iVersionMajor,
        iVersionMinor
);

;#END_EDIT_BLOCK END_FUNCTION

#END_OF_IEC_PART

@Puma @IecEditor 6 68 @Pou 25
@@@BEG_Comment@@@
@h    ! WARNING !
@h    The Kemro K2 system (including software) only meets category B according to EN 954-1,
@h    thus it is not intended for usage in safety-relevant control applications in the field
@h    of personal safety (e.g. emergency stop).
@h    To implement potentially necessary safety-relevant control tasks, always use additional
@h    external safety devices that are intended for the particular purpose, and meet the necessary
@h    functional safety.
@h    For further information see EN 954-1 (EN ISO 13849-1) and/or the K2-x00 user manual, chapter
@h    "CE conformity, directives and standards".

Create empty catalog entry for HMI.Style version info because there is no possibility to create catalog nodes
in HMI.Style. Version Info will be written by HMI.Style at startup.
@@@END_Comment@@@

@BEG_Contents

@BEG_Func
@RT(17)FuncTreeContainer
1
@Var @RT(22)FWriteComponentVersion @RT(0) @T @T @DERIVED 0 @F @RT(8)FUNCTION @F
@T
@BEG_Attrib
0 @RT(0) @RT(0)
@END_Attrib
1 1 @F @F @F @F

@END_Func

@BEG_Const
@RT(18)ConstTreeContainer
0
@END_Const

@BEG_Export

@BEG_Kind
@FUNCTION @RT(22)FCreateHMIStyleVersion @STRUCTURED_TEXT
@RT(4)BOOL @RT(0) @RT(0)
@END_Kind

@BEG_Dcl
@RT(16)DclTreeContainer
5
@Var @RT(14)sComponentName @RT(0) @T @F @DT @RT(11)STRING(255) @RT(0) @T @T @STRING 0 @F @RT(3)255 @F
@F @F
@T
@BEG_Attrib
3 @RT(19)'KePlast.HMI.Style' @RT(0) @RT(0)
@END_Attrib
1 15 @F @F @F @F

@Var @RT(16)iComponentNumber @RT(0) @T @F @DT @RT(4)DINT @RT(0) @T @T @BASIC 0 @F
@F @F
@T
@BEG_Attrib
3 @RT(1)0 @RT(0) @RT(0)
@END_Attrib
1 15 @F @F @F @F

@Var @RT(14)sVersionString @RT(0) @T @F @DT @RT(11)STRING(255) @RT(0) @T @T @STRING 0 @F @RT(3)255 @F
@F @F
@T
@BEG_Attrib
3 @RT(2)'' @RT(0) @RT(0)
@END_Attrib
1 15 @F @F @F @F

@Var @RT(13)iVersionMajor @RT(0) @T @F @DT @RT(4)DINT @RT(0) @T @T @BASIC 0 @F
@F @F
@T
@BEG_Attrib
3 @RT(1)0 @RT(0) @RT(0)
@END_Attrib
1 15 @F @F @F @F

@Var @RT(13)iVersionMinor @RT(0) @T @F @DT @RT(4)DINT @RT(0) @T @T @BASIC 0 @F
@F @F
@T
@BEG_Attrib
3 @RT(1)0 @RT(0) @RT(0)
@END_Attrib
1 15 @F @F @F @F

@END_Dcl

@END_Export

@BEG_Body
@TL(13)
(**************************************** WARNING ********************************************
 *** The KEBA Kemro K2 System including software is not intended for safety control tasks! ***
 ***                       For further information see Comment tab!                        ***
 *********************************************************************************************)

FCreateHMIStyleVersion := FWriteComponentVersion(
        sComponentName,
        iComponentNumber,
        sVersionString,
        iVersionMajor,
        iVersionMinor
);

@END_Body

@END_Contents

(* ---- FCreateIECVersion.pu ---- *)
(*
@h    ! WARNING !
@h    The Kemro K2 system (including software) only meets category B according to EN 954-1,
@h    thus it is not intended for usage in safety-relevant control applications in the field
@h    of personal safety (e.g. emergency stop).
@h    To implement potentially necessary safety-relevant control tasks, always use additional
@h    external safety devices that are intended for the particular purpose, and meet the necessary
@h    functional safety.
@h    For further information see EN 954-1 (EN ISO 13849-1) and/or the K2-x00 user manual, chapter
@h    "CE conformity, directives and standards".

this file is automatically created by clearcase makebaseline
and contains versioninformation of component
*)

IMPORT_OVER_LISTFILE
 FWriteComponentVersion

END_IMPORT

FUNCTION FCreateIECVersion : BOOL #DUMMY_EDIT_BLOCK

VAR CONSTANT
 sComponentName : STRING(255) := 'KePlast.IEC';
 iComponentNumber : DINT := 0;
 sVersionString : STRING(255) := 'KePlast.IEC_01.56';
 iVersionMajor : DINT := 1;
 iVersionMinor : DINT := 56;
END_VAR
#BEGIN_EDIT_BLOCK
(**************************************** WARNING ********************************************
 *** The KEBA Kemro K2 System including software is not intended for safety control tasks! ***
 ***                       For further information see Comment tab!                        ***
 *********************************************************************************************)

FCreateIECVersion := FWriteComponentVersion(
        sComponentName,
        iComponentNumber,
        sVersionString,
        iVersionMajor,
        iVersionMinor
);

;#END_EDIT_BLOCK END_FUNCTION

#END_OF_IEC_PART

@Puma @IecEditor 6 68 @Pou 25
@@@BEG_Comment@@@
@h    ! WARNING !
@h    The Kemro K2 system (including software) only meets category B according to EN 954-1,
@h    thus it is not intended for usage in safety-relevant control applications in the field
@h    of personal safety (e.g. emergency stop).
@h    To implement potentially necessary safety-relevant control tasks, always use additional
@h    external safety devices that are intended for the particular purpose, and meet the necessary
@h    functional safety.
@h    For further information see EN 954-1 (EN ISO 13849-1) and/or the K2-x00 user manual, chapter
@h    "CE conformity, directives and standards".

this file is automatically created by clearcase makebaseline
and contains versioninformation of component
@@@END_Comment@@@

@BEG_Contents

@BEG_Func
@RT(17)FuncTreeContainer
1
@Var @RT(22)FWriteComponentVersion @RT(0) @T @F @DT @RT(0) @RT(0) @T @T @UNKNOWN 0 @F
@F @F
@T
@BEG_Attrib
0 @RT(0) @RT(0)
@END_Attrib
1 1 @F @F @F @F

@END_Func

@BEG_Const
@RT(18)ConstTreeContainer
0
@END_Const

@BEG_Export

@BEG_Kind
@FUNCTION @RT(17)FCreateIECVersion @STRUCTURED_TEXT
@RT(4)BOOL @RT(0) @RT(0)
@END_Kind

@BEG_Dcl
@RT(16)DclTreeContainer
5
@Var @RT(14)sComponentName @RT(0) @T @F @DT @RT(11)STRING(255) @RT(0) @T @T @STRING 0 @F @RT(3)255 @F
@F @F
@T
@BEG_Attrib
3 @RT(13)'KePlast.IEC' @RT(0) @RT(0)
@END_Attrib
1 15 @F @F @F @F

@Var @RT(16)iComponentNumber @RT(0) @T @F @DT @RT(4)DINT @RT(0) @T @T @BASIC 0 @F
@F @F
@T
@BEG_Attrib
3 @RT(1)0 @RT(0) @RT(0)
@END_Attrib
1 15 @F @F @F @F

@Var @RT(14)sVersionString @RT(0) @T @F @DT @RT(11)STRING(255) @RT(0) @T @T @STRING 0 @F @RT(3)255 @F
@F @F
@T
@BEG_Attrib
3 @RT(19)'KePlast.IEC_01.56' @RT(0) @RT(0)
@END_Attrib
1 15 @F @F @F @F

@Var @RT(13)iVersionMajor @RT(0) @T @F @DT @RT(4)DINT @RT(0) @T @T @BASIC 0 @F
@F @F
@T
@BEG_Attrib
3 @RT(1)1 @RT(0) @RT(0)
@END_Attrib
1 15 @F @F @F @F

@Var @RT(13)iVersionMinor @RT(0) @T @F @DT @RT(4)DINT @RT(0) @T @T @BASIC 0 @F
@F @F
@T
@BEG_Attrib
3 @RT(2)56 @RT(0) @RT(0)
@END_Attrib
1 15 @F @F @F @F

@END_Dcl

@END_Export

@BEG_Body
@TL(13)
(**************************************** WARNING ********************************************
 *** The KEBA Kemro K2 System including software is not intended for safety control tasks! ***
 ***                       For further information see Comment tab!                        ***
 *********************************************************************************************)

FCreateIECVersion := FWriteComponentVersion(
        sComponentName,
        iComponentNumber,
        sVersionString,
        iVersionMajor,
        iVersionMinor
);

@END_Body

@END_Contents

(* ---- FCreateSystemName.pu ---- *)
IMPORT_OVER_LISTFILE
 FGetSystemName
, KCAT_HandleData
, KCAT_Status

END_IMPORT

FUNCTION FCreateSystemName : BOOL #DUMMY_EDIT_BLOCK

VAR
 HandleData : KCAT_HandleData;
 sTmp : STRING(255);
 Status : KCAT_Status;
END_VAR
#BEGIN_EDIT_BLOCK
(**************************************** WARNING ********************************************
 *** The KEBA Kemro K2 System including software is not intended for safety control tasks! ***
 ***                       For further information see Comment tab!                        ***
 *********************************************************************************************)

sTmp := "Application";

HandleData := KCAT_GetHandle(sTmp);
IF HandleData.Status <> KCAT_Status_OK THEN
    RETURN;
END_IF;

HandleData := KCAT_AddDir(HandleData.Handle, "KePlast");
IF HandleData.Status <> KCAT_Status_OK THEN
    RETURN;
END_IF;

sTmp := FGetSystemName();
Status := KCAT_AddValue(HandleData.Handle, "systemName", KCAT_Type_STRING, sTmp);
IF Status <> KCAT_Status_OK THEN
    RETURN;
END_IF;

FCreateSystemName := TRUE;

;#END_EDIT_BLOCK END_FUNCTION

#END_OF_IEC_PART

@Puma @IecEditor 6 80 @Pou 25
@@@BEG_Comment@@@

@@@END_Comment@@@

@BEG_Contents

@BEG_Func
@RT(17)FuncTreeContainer
1
@Var @RT(14)FGetSystemName @RT(0) @T @T @DERIVED 0 @F @RT(21)FUNCTION : STRING(31) @F
@T
@BEG_Attrib
0 @RT(0) @RT(0)
@END_Attrib
1 1 @F @F @F @F

@END_Func

@BEG_Const
@RT(18)ConstTreeContainer
0
@END_Const

@BEG_Export

@BEG_Kind
@FUNCTION @RT(17)FCreateSystemName @STRUCTURED_TEXT
@RT(4)BOOL @RT(0) @RT(0)
@END_Kind

@BEG_Dcl
@RT(16)DclTreeContainer
3
@Var @RT(10)HandleData @RT(0) @T @T @DERIVED 0 @F @RT(15)KCAT_HandleData @F
@T
@BEG_Attrib
3 @RT(0) @RT(0) @RT(0)
@END_Attrib
1 0 @F @F @F @F

@Var @RT(4)sTmp @RT(0) @T @F @DT @RT(11)STRING(255) @RT(0) @T @T @STRING 0 @F @RT(3)255 @F
@F @F
@T
@BEG_Attrib
3 @RT(0) @RT(0) @RT(0)
@END_Attrib
1 0 @F @F @F @F

@Var @RT(6)Status @RT(0) @T @T @DERIVED 0 @F @RT(11)KCAT_Status @F
@T
@BEG_Attrib
3 @RT(0) @RT(0) @RT(0)
@END_Attrib
1 0 @F @F @F @F

@END_Dcl

@END_Export

@BEG_Body
@TL(26)
(**************************************** WARNING ********************************************
 *** The KEBA Kemro K2 System including software is not intended for safety control tasks! ***
 ***                       For further information see Comment tab!                        ***
 *********************************************************************************************)

sTmp := "Application";

HandleData := KCAT_GetHandle(sTmp);
IF HandleData.Status <> KCAT_Status_OK THEN
    RETURN;
END_IF;

HandleData := KCAT_AddDir(HandleData.Handle, "KePlast");
IF HandleData.Status <> KCAT_Status_OK THEN
    RETURN;
END_IF;

sTmp := FGetSystemName();
Status := KCAT_AddValue(HandleData.Handle, "systemName", KCAT_Type_STRING, sTmp);
IF Status <> KCAT_Status_OK THEN
    RETURN;
END_IF;

FCreateSystemName := TRUE;

@END_Body

@END_Contents

(* ---- FGetSystemName.pu ---- *)
FUNCTION FGetSystemName : STRING(31) #DUMMY_EDIT_BLOCK

VAR CONSTANT
 sSYSTEMNAME : STRING(31) := 'KePlast i2980';
END_VAR
#BEGIN_EDIT_BLOCK
FGetSystemName := sSYSTEMNAME;

;#END_EDIT_BLOCK END_FUNCTION

#END_OF_IEC_PART

@Puma @IecEditor 6 80 @Pou 25
@@@BEG_Comment@@@

@@@END_Comment@@@

@BEG_Contents

@BEG_Func
@RT(17)FuncTreeContainer
0
@END_Func

@BEG_Const
@RT(18)ConstTreeContainer
0
@END_Const

@BEG_Export

@BEG_Kind
@FUNCTION @RT(14)FGetSystemName @STRUCTURED_TEXT
@RT(10)STRING(31) @RT(0) @RT(0)
@END_Kind

@BEG_Dcl
@RT(16)DclTreeContainer
1
@Var @RT(11)sSYSTEMNAME @RT(0) @T @F @DT @RT(10)STRING(31) @RT(0) @T @T @STRING 0 @F @RT(2)31 @F
@F @F
@T
@BEG_Attrib
3 @RT(15)'KePlast i2980' @RT(0) @RT(0)
@END_Attrib
1 15 @F @F @F @F

@END_Dcl

@END_Export

@BEG_Body
@TL(2)
FGetSystemName := sSYSTEMNAME;

@END_Body

@END_Contents

(* ---- ABDeviceRegistration.pu ---- *)
(*
@h    ! WARNING !
@h    The Kemro K2 system (including software) only meets category B according to EN 954-1,
@h    thus it is not intended for usage in safety-relevant control applications in the field
@h    of personal safety (e.g. emergency stop).
@h    To implement potentially necessary safety-relevant control tasks, always use additional
@h    external safety devices that are intended for the particular purpose, and meet the necessary
@h    functional safety.
@h    For further information see EN 954-1 (EN ISO 13849-1) and/or the K2-x00 user manual, chapter
@h    "CE conformity, directives and standards".

This AB collects the deviceregistration events which are sent by every FU during iec-initialisation.
The registered devices are written into the array sv_NumberOfDevices to have the possibility to check
how many devices of a component are available on the system.
*)

IMPORT_OVER_LISTFILE
 SET_ALARM
, STOP_PROCESS_ALGORITHM
, cMaxCompId
, cCompPump
, tyNumberOfDevices
, tevDeviceRegister
, tevDeviceRegisterData
, tyRegisteredDevices
, ABRegisterDelay

END_IMPORT

ALGORITHM_BLOCK ABDeviceRegistration #DUMMY_EDIT_BLOCK

SYSTEM_VAR
 sv_NumberOfDevices : tyNumberOfDevices;
 sv_iDevicesToRegister : DINT (* Number of devices registered *);
 sv_bDeviceRegisterDone : BOOL;
END_VAR

SYSTEM_OBJECT
 EV_Task_3 : TASK;
 erMultipleDeviceReg : ALARM;
 erMaxDeviceIndexExeeded : ALARM;
 erMaxCompIdExeeded : ALARM;
 evDeviceRegister : tevDeviceRegister;
 Task10ms : TASK;
 erDeviceReg : ALARM;
 erTooManyPumpsRegistered : ALARM;
END_OBJECT

VAR
 m_iRegistrationCounter : DINT;
END_VAR

(*
This algo receives the registration event from each device.
To prevent from programming mistakes following checks are done:
  - overrun of maximum Component-ID
  - overrun of maximum Device-index
  - occurence of multiple registration of any device
*)

EVENT_ALGORITHM evaDeviceRegister ON EV_Task_3 WITH evDeviceRegister

VAR_INPUT
 evDeviceRegisterData : tevDeviceRegisterData;
END_VAR

VAR
 registeredDevices : tyRegisteredDevices;
 dummy : DINT;
END_VAR
#BEGIN_EDIT_BLOCK
(**************************************** WARNING ********************************************
 *** The KEBA Kemro K2 System including software is not intended for safety control tasks! ***
 ***                       For further information see Comment tab!                        ***
 *********************************************************************************************)

//receiving device registrationevents

IF evDeviceRegisterData.DeviceId.CompId > cMaxCompId THEN
    SET_ALARM(Name := erMaxCompIdExeeded,
                SubID1 := cMaxCompId);
    //registration error: stop device registration
    STOP_PROCESS_ALGORITHM(paDeviceRegister);
    RETURN;
END_IF;

IF evDeviceRegisterData.DeviceId.IndexId > cMaxDeviceIndex THEN
    SET_ALARM(Name := erMaxDeviceIndexExeeded,
                SubID1 := evDeviceRegisterData.DeviceId.CompId,
                SubID2 := cMaxDeviceIndex);
    //registration error: stop device registration
    STOP_PROCESS_ALGORITHM(paDeviceRegister);
    RETURN;
END_IF;

//check limit of allowed pump - FU´s
IF evDeviceRegisterData.DeviceId.CompId = cCompPump THEN
    //limit of pumps already reached
    IF sv_NumberOfDevices[cCompPump] = cMaxNrOfPumps THEN
        SET_ALARM(Name := erTooManyPumpsRegistered);
        STOP_PROCESS_ALGORITHM(paDeviceRegister);
        RETURN;
    END_IF;
END_IF;

//checking for multiple registrations
IF NOT registeredDevices[evDeviceRegisterData.DeviceId.CompId]
                        [evDeviceRegisterData.DeviceId.IndexId] THEN
    m_iRegistrationCounter := m_iRegistrationCounter + 1;

    // incrementing registrationcounter for each compId
    sv_NumberOfDevices[evDeviceRegisterData.DeviceId.CompId] :=
    sv_NumberOfDevices[evDeviceRegisterData.DeviceId.CompId] + 1;

    // remembering that the device is already registered
    registeredDevices[evDeviceRegisterData.DeviceId.CompId]
                        [evDeviceRegisterData.DeviceId.IndexId] := TRUE;
ELSE
   // Device has been registered multiple
   SET_ALARM(Name := erMultipleDeviceReg,
            SubID1 := evDeviceRegisterData.DeviceId.CompId,
            SubID2 := evDeviceRegisterData.DeviceId.IndexId);

   dummy := Print("Multiple device registration: %d.%d",
                  evDeviceRegisterData.DeviceId.CompId,
                  evDeviceRegisterData.DeviceId.IndexId);

   //registration error: stop device registration
   STOP_PROCESS_ALGORITHM(paDeviceRegister);
END_IF;

;#END_EDIT_BLOCK END_ALGORITHM

(*
Waits for the registration process and sets the sv_bInitStart flag if registration succeeds.
Registration is ready if the sv_iDevicesRegistered is equal to the running registration counter.
The start-delay is done to give the devices time for incrementing sv_iDevicesRegistered.

*)

PROCESS_ALGORITHM paDeviceRegister ON Task10ms AUTOSTART

VAR
 abRegisterDelay : ABRegisterDelay;
END_VAR

(* IecGraph-Code *)

(* init step *)
INITIAL_STEP DELAY:
END_STEP

(* steps *)
STEP REG_ACTIVE:
END_STEP

STEP REG_ERROR:
Action5 (P);
END_STEP

ACTION Action5: #BEGIN_EDIT_BLOCK
SET_ALARM(Name := erDeviceReg);

;#END_EDIT_BLOCK END_ACTION (*Action5*)
STEP REG_FINISHED:
aRegistrationFinished (P);
END_STEP

ACTION aRegistrationFinished: #BEGIN_EDIT_BLOCK
// Device registration finished
sv_bDeviceRegisterDone := TRUE;

// reset delaytime generator
abRegisterDelay.aReset();

;#END_EDIT_BLOCK END_ACTION (*aRegistrationFinished*)
STEP END:
Action8 (P);
END_STEP

ACTION Action8: #BEGIN_EDIT_BLOCK
STOP_PROCESS_ALGORITHM();

;#END_EDIT_BLOCK END_ACTION (*Action8*)

(* transitions *)
TRANSITION Trans1 (* Trans1 *) FROM DELAY TO REG_ACTIVE :=  #BEGIN_EDIT_BLOCK
DELAY.T >= T#200ms
;#END_EDIT_BLOCK
(*give the devices time to increment sv_iDevicesToRegister*)
END_TRANSITION

TRANSITION Trans2 (* Trans2 *) FROM REG_ACTIVE TO REG_FINISHED :=  #BEGIN_EDIT_BLOCK
m_iRegistrationCounter =
sv_iDevicesToRegister
;#END_EDIT_BLOCK
END_TRANSITION

TRANSITION Trans3 (* Trans3 *) FROM REG_ACTIVE TO REG_ERROR :=  #BEGIN_EDIT_BLOCK
m_iRegistrationCounter >
sv_iDevicesToRegister

;#END_EDIT_BLOCK
END_TRANSITION

GO_ON_TRANSITION Trans9 (* Trans9 *) FROM REG_ERROR TO END :=  #BEGIN_EDIT_BLOCK
TRUE
;#END_EDIT_BLOCK
END_TRANSITION

GO_ON_TRANSITION Trans10 (* Trans10 *) FROM REG_FINISHED TO END :=  #BEGIN_EDIT_BLOCK
TRUE
;#END_EDIT_BLOCK
END_TRANSITION

(* end IecGraph-Code *)
(* sfc-code *)
(* end sfc-code *)

END_ALGORITHM

END_ALGORITHM_BLOCK

#END_OF_IEC_PART

@Puma @IecEditor 6 80 @Pou 25
@@@BEG_Comment@@@
@h    ! WARNING !
@h    The Kemro K2 system (including software) only meets category B according to EN 954-1,
@h    thus it is not intended for usage in safety-relevant control applications in the field
@h    of personal safety (e.g. emergency stop).
@h    To implement potentially necessary safety-relevant control tasks, always use additional
@h    external safety devices that are intended for the particular purpose, and meet the necessary
@h    functional safety.
@h    For further information see EN 954-1 (EN ISO 13849-1) and/or the K2-x00 user manual, chapter
@h    "CE conformity, directives and standards".

This AB collects the deviceregistration events which are sent by every FU during iec-initialisation.
The registered devices are written into the array sv_NumberOfDevices to have the possibility to check
how many devices of a component are available on the system.
@@@END_Comment@@@

@BEG_Contents

@BEG_Func
@RT(17)FuncTreeContainer
2
@Var @RT(9)SET_ALARM @RT(0) @T @T @DERIVED 0 @F @RT(23)KEBA_STANDARD_PROCEDURE @F
@T
@BEG_Attrib
0 @RT(0) @RT(0)
@END_Attrib
1 1 @F @F @F @F

@Var @RT(22)STOP_PROCESS_ALGORITHM @RT(0) @T @T @DERIVED 0 @F @RT(23)KEBA_STANDARD_PROCEDURE @F
@T
@BEG_Attrib
0 @RT(0) @RT(0)
@END_Attrib
1 1 @F @F @F @F

@END_Func

@BEG_Const
@RT(18)ConstTreeContainer
2
@Var @RT(10)cMaxCompId @RT(0) @T @F @DT @RT(4)DINT @RT(0) @T @T @BASIC 0 @F
@F @F
@T
@BEG_Attrib
0 @RT(3)250 @RT(21)maximum Component ID
@END_Attrib
1 1 @F @F @F @F

@Var @RT(9)cCompPump @RT(0) @T @F @DT @RT(4)DINT @RT(0) @T @T @BASIC 0 @F
@F @F
@T
@BEG_Attrib
0 @RT(3)113 @RT(14)Component Pump
@END_Attrib
1 1 @F @F @F @F

@END_Const

@BEG_Export

@BEG_Kind
@ALGORITHM_BLOCK @RT(20)ABDeviceRegistration @STRUCTURED_TEXT
@RT(0) @RT(0) @RT(0)
@END_Kind

@BEG_Dcl
@RT(16)DclTreeContainer
12
@Var @RT(9)EV_Task_3 @RT(0) @T @T @RENAMED 0 @T @T @DT @RT(4)TASK @RT(0) @T @T @BASIC 0 @F
@F @F
@T
@BEG_Attrib
3 @RT(0) @RT(0) @RT(0)
@END_Attrib
1 7 @F @F @F @F

@Var @RT(19)erMultipleDeviceReg @RT(0) @T @F @DT @RT(5)ALARM @RT(0) @T @T @BASIC 0 @F
@F @F
@T
@BEG_Attrib
3 @RT(0) @RT(0) @RT(0)
@END_Attrib
1 7 @F @F @F @F

@Var @RT(23)erMaxDeviceIndexExeeded @RT(0) @T @F @DT @RT(5)ALARM @RT(0) @T @T @BASIC 0 @F
@F @F
@T
@BEG_Attrib
3 @RT(0) @RT(0) @RT(0)
@END_Attrib
1 7 @F @F @F @F

@Var @RT(18)erMaxCompIdExeeded @RT(0) @T @F @DT @RT(5)ALARM @RT(0) @T @T @BASIC 0 @F
@F @F
@T
@BEG_Attrib
3 @RT(0) @RT(0) @RT(0)
@END_Attrib
1 7 @F @F @F @F

@Var @RT(18)sv_NumberOfDevices @RT(0) @T @T @DERIVED 0 @T @T @DT @RT(17)tyNumberOfDevices @RT(0) @T @T @UNKNOWN 0 @F
@F @F
@T
@BEG_Attrib
3 @RT(0) @RT(0) @RT(0)
@END_Attrib
1 8 @F @F @F @F

@Var @RT(21)sv_iDevicesToRegister @RT(0) @T @F @DT @RT(4)DINT @RT(0) @T @T @BASIC 0 @F
@F @F
@T
@BEG_Attrib
3 @RT(0) @RT(28)Number of devices registered @RT(0)
@END_Attrib
1 8 @F @F @F @F

@Var @RT(16)evDeviceRegister @RT(0) @T @T @RENAMED 0 @T @T @DT @RT(17)tevDeviceRegister @RT(0) @T @T @UNKNOWN 0 @F
@F @F
@T
@BEG_Attrib
3 @RT(0) @RT(0) @RT(0)
@END_Attrib
1 7 @F @F @F @F

@Var @RT(22)m_iRegistrationCounter @RT(0) @T @F @DT @RT(4)DINT @RT(0) @T @T @BASIC 0 @F
@F @F
@T
@BEG_Attrib
3 @RT(0) @RT(0) @RT(0)
@END_Attrib
1 0 @F @F @F @F

@Var @RT(8)Task10ms @RT(0) @T @T @RENAMED 0 @T @T @DT @RT(4)TASK @RT(0) @T @T @BASIC 0 @F
@F @F
@T
@BEG_Attrib
3 @RT(0) @RT(0) @RT(0)
@END_Attrib
1 7 @F @F @F @F

@Var @RT(11)erDeviceReg @RT(0) @T @F @DT @RT(5)ALARM @RT(0) @T @T @BASIC 0 @F
@F @F
@T
@BEG_Attrib
3 @RT(0) @RT(0) @RT(0)
@END_Attrib
1 7 @F @F @F @F

@Var @RT(22)sv_bDeviceRegisterDone @RT(0) @T @F @DT @RT(4)BOOL @RT(0) @T @T @BASIC 0 @F
@F @F
@T
@BEG_Attrib
3 @RT(0) @RT(0) @RT(0)
@END_Attrib
1 8 @F @F @F @F

@Var @RT(24)erTooManyPumpsRegistered @RT(0) @T @F @DT @RT(5)ALARM @RT(0) @T @T @BASIC 0 @F
@F @F
@T
@BEG_Attrib
3 @RT(0) @RT(0) @RT(0)
@END_Attrib
1 7 @F @F @F @F

@END_Dcl

@END_Export

@BEG_Body

2

@BEG_Export

@BEG_Algo
@EVENT_ALGORITHM @RT(17)evaDeviceRegister @STRUCTURED_TEXT
@RT(0) @RT(16)evDeviceRegister @RT(9)EV_Task_3 @F @F
@END_Algo

@BEG_Dcl
@RT(16)DclTreeContainer
3
@Var @RT(20)evDeviceRegisterData @RT(0) @T @T @DERIVED 0 @F @RT(21)tevDeviceRegisterData @F
@T
@BEG_Attrib
3 @RT(0) @RT(0) @RT(0)
@END_Attrib
1 1 @F @F @F @F

@Var @RT(17)registeredDevices @RT(0) @T @T @DERIVED 0 @T @T @DT @RT(19)tyRegisteredDevices @RT(0) @T @T @UNKNOWN 0 @F
@F @F
@T
@BEG_Attrib
3 @RT(0) @RT(0) @RT(0)
@END_Attrib
1 0 @F @F @F @F

@Var @RT(5)dummy @RT(0) @T @F @DT @RT(4)DINT @RT(0) @T @T @BASIC 0 @F
@F @F
@T
@BEG_Attrib
3 @RT(0) @RT(0) @RT(0)
@END_Attrib
1 0 @F @F @F @F

@END_Dcl

@END_Export

@BEG_Export

@BEG_Algo
@PROCESS_ALGORITHM @RT(16)paDeviceRegister @SEQUENTIAL_FLOW_CHART
@RT(0) @RT(0) @RT(8)Task10ms @T @F
@END_Algo

@BEG_Dcl
@RT(16)DclTreeContainer
1
@Var @RT(15)abRegisterDelay @RT(0) @T @T @DERIVED 0 @T @T @DT @RT(15)ABRegisterDelay @RT(0) @T @T @UNKNOWN 0 @F
@F @F
@T
@BEG_Attrib
3 @RT(0) @RT(0) @RT(0)
@END_Attrib
1 0 @F @F @F @F

@END_Dcl

@END_Export

@BEG_Body
@TL(60)
(**************************************** WARNING ********************************************
 *** The KEBA Kemro K2 System including software is not intended for safety control tasks! ***
 ***                       For further information see Comment tab!                        ***
 *********************************************************************************************)

//receiving device registrationevents

IF evDeviceRegisterData.DeviceId.CompId > cMaxCompId THEN
    SET_ALARM(Name := erMaxCompIdExeeded,
                SubID1 := cMaxCompId);
    //registration error: stop device registration
    STOP_PROCESS_ALGORITHM(paDeviceRegister);
    RETURN;
END_IF;

IF evDeviceRegisterData.DeviceId.IndexId > cMaxDeviceIndex THEN
    SET_ALARM(Name := erMaxDeviceIndexExeeded,
                SubID1 := evDeviceRegisterData.DeviceId.CompId,
                SubID2 := cMaxDeviceIndex);
    //registration error: stop device registration
    STOP_PROCESS_ALGORITHM(paDeviceRegister);
    RETURN;
END_IF;

//check limit of allowed pump - FU´s
IF evDeviceRegisterData.DeviceId.CompId = cCompPump THEN
    //limit of pumps already reached
    IF sv_NumberOfDevices[cCompPump] = cMaxNrOfPumps THEN
        SET_ALARM(Name := erTooManyPumpsRegistered);
        STOP_PROCESS_ALGORITHM(paDeviceRegister);
        RETURN;
    END_IF;
END_IF;

//checking for multiple registrations
IF NOT registeredDevices[evDeviceRegisterData.DeviceId.CompId]
                        [evDeviceRegisterData.DeviceId.IndexId] THEN
    m_iRegistrationCounter := m_iRegistrationCounter + 1;

    // incrementing registrationcounter for each compId
    sv_NumberOfDevices[evDeviceRegisterData.DeviceId.CompId] :=
    sv_NumberOfDevices[evDeviceRegisterData.DeviceId.CompId] + 1;

    // remembering that the device is already registered
    registeredDevices[evDeviceRegisterData.DeviceId.CompId]
                        [evDeviceRegisterData.DeviceId.IndexId] := TRUE;
ELSE
   // Device has been registered multiple
   SET_ALARM(Name := erMultipleDeviceReg,
            SubID1 := evDeviceRegisterData.DeviceId.CompId,
            SubID2 := evDeviceRegisterData.DeviceId.IndexId);

   dummy := Print("Multiple device registration: %d.%d",
                  evDeviceRegisterData.DeviceId.CompId,
                  evDeviceRegisterData.DeviceId.IndexId);

   //registration error: stop device registration
   STOP_PROCESS_ALGORITHM(paDeviceRegister);
END_IF;

@END_Body

@@@BEG_Comment@@@
@TL(5)
This algo receives the registration event from each device.
To prevent from programming mistakes following checks are done:
  - overrun of maximum Component-ID
  - overrun of maximum Device-index
  - occurence of multiple registration of any device
@@@END_Comment@@@

@BEG_SfcBody
9 9 11

@BEG_SfcData 2
@StepSeq @RT(4)sseq @F 7
@Step @RT(5)DELAY @F @T @F @F @RT(0) @F
@AcbCont @RT(7)unnamed @F 0

@Trans @RT(6)Trans1 @F @T @F @F @T @T @TL(2)
DELAY.T >= T#200ms

@RT(6)Trans1 @T @TL(1)
give the devices time to increment sv_iDevicesToRegister

@Step @RT(10)REG_ACTIVE @F @F @F @F @RT(0) @F
@AcbCont @RT(7)unnamed @F 0

@AltBranch @RT(3)alt @F 2
@TransSeq @RT(4)tseq @F 1
@Trans @RT(6)Trans2 @F @T @F @F @T @T @TL(3)
m_iRegistrationCounter =
sv_iDevicesToRegister

@RT(6)Trans2 @F

@TransSeq @RT(4)tseq @F 4
@Trans @RT(6)Trans3 @F @T @F @F @T @T @TL(4)
m_iRegistrationCounter >
sv_iDevicesToRegister

@RT(6)Trans3 @F
@Step @RT(9)REG_ERROR @F @F @F @F @RT(0) @F
@AcbCont @RT(7)unnamed @F 1
@Acb @RT(7)Action5 @F @T @RT(1)P @RT(0) @F @F @T @TL(2)
SET_ALARM(Name := erDeviceReg);

@F

@Trans @RT(6)Trans9 @F @T @F @F @T @F @TL(2)
TRUE

@RT(6)Trans9 @F
@Goto @RT(3)END @F @F

@Step @RT(12)REG_FINISHED @F @F @F @F @RT(0) @F
@AcbCont @RT(7)unnamed @F 1
@Acb @RT(21)aRegistrationFinished @F @T @RT(1)P @RT(0) @F @F @T @TL(6)
// Device registration finished
sv_bDeviceRegisterDone := TRUE;

// reset delaytime generator
abRegisterDelay.aReset();

@F

@Trans @RT(7)Trans10 @F @T @F @F @T @F @TL(2)
TRUE

@RT(7)Trans10 @F
@Step @RT(3)END @F @F @T @F @RT(0) @F
@AcbCont @RT(7)unnamed @F 1
@Acb @RT(7)Action8 @F @T @RT(1)P @RT(0) @F @F @T @TL(2)
STOP_PROCESS_ALGORITHM();

@F

@END_SfcData
@SaActions 0
@SaTrans 0
@SaExits 0
@END_SfcBody

@@@BEG_Comment@@@
@TL(4)
Waits for the registration process and sets the sv_bInitStart flag if registration succeeds.
Registration is ready if the sv_iDevicesRegistered is equal to the running registration counter.
The start-delay is done to give the devices time for incrementing sv_iDevicesRegistered.

@@@END_Comment@@@
@END_Body

@END_Contents
